// TIA Portal project "bascule_de_controle" (V15)

(* hardware
DEVICE "Station S7-1200_1"  S7-1200 Station
   slot 0: "Châssis_0"  S7-1200 Rack  Rack  V1.0
   slot 1: "PLC_1"  CPU 1215C AC/DC/Rly  6ES7 215-1BG40-0XB0  V4.2
DEVICE "HMI_1"  KTP700 Basic PN
   slot 0: "HMI_1"  KTP700 Basic PN  6AV2 123-2GB03-0AX0  15.0.0.0
   slot 1: "HMI_RT_1"  KTP700 Basic PN  6AV2 123-2GB03-0AX0  15.0.0.0
   slot 5: "HMI_1.IE_CP_1"  PROFINET Interface  15.0.0.0
      slot 1: "Interface PROFINET_1"  PROFINET Interface
         slot 1: "Port_1"  Port
*)

// ===== PLC "PLC_1"  CPU 1215C AC/DC/Rly =====

VAR_GLOBAL   // PLC tag table "Table de variables standard"
   "System_Byte" AT %MB1 : Byte;
   "FirstScan" AT %M1.0 : Bool;
   "DiagStatusUpdate" AT %M1.1 : Bool;
   "AlwaysTRUE" AT %M1.2 : Bool;
   "AlwaysFALSE" AT %M1.3 : Bool;
   "Clock_Byte" AT %MB0 : Byte;
   "Clock_10Hz" AT %M0.0 : Bool;
   "Clock_5Hz" AT %M0.1 : Bool;
   "Clock_2.5Hz" AT %M0.2 : Bool;
   "Clock_2Hz" AT %M0.3 : Bool;
   "Clock_1.25Hz" AT %M0.4 : Bool;
   "Clock_1Hz" AT %M0.5 : Bool;
   "Clock_0.625Hz" AT %M0.6 : Bool;
   "Clock_0.5Hz" AT %M0.7 : Bool;
   "temps_ecoulées" AT %M5.1 : Bool;
   "compter" AT %MW7 : Int;
   "temps_ecoulés" AT %M5.0 : Bool;
   "pesage" AT %MW3 : Word;
   "nbre_bac" AT %MW10 : Int;
   "C_OK" AT %M9.0 : Bool;
   "ENABLE" AT %M9.1 : Bool;
   "depart" AT %Q0.7 : Bool;
END_VAR

VAR_GLOBAL   // PLC tag table "variables_pfa"
   "dcy" AT %I0.0 : Bool;
   "S0" AT %I0.1 : Bool;
   "S1" AT %I0.2 : Bool;
   "EB" AT %I0.3 : Bool;
   "SB" AT %I0.4 : Bool;
   "Tv" AT %I0.5 : Bool;
   "Tf" AT %I0.6 : Bool;
   "C10" AT %I0.7 : Bool;
   "C11" AT %I1.0 : Bool;
   "C20" AT %I1.1 : Bool;
   "C21" AT %I1.2 : Bool;
   "X0" AT %M2.0 : Bool;
   "X1" AT %M2.1 : Bool;
   "X2" AT %M2.2 : Bool;
   "X3" AT %M2.3 : Bool;
   "X4" AT %M2.4 : Bool;
   "X5" AT %M2.5 : Bool;
   "X6" AT %M2.6 : Bool;
   "X7" AT %M2.7 : Bool;
   "X8" AT %M3.0 : Bool;
   "X9" AT %M3.1 : Bool;
   "X10" AT %M3.2 : Bool;
   "X11" AT %M3.3 : Bool;
   "KM1" AT %Q0.0 : Bool;
   "H1" AT %Q0.1 : Bool;
   "BP" AT %Q0.2 : Bool;
   "SV1" AT %Q0.3 : Bool;
   "RV1" AT %Q0.4 : Bool;
   "SV2" AT %Q0.5 : Bool;
   "RV2" AT %Q0.6 : Bool;
   "RA" AT %I1.3 : Bool;
   "alarm_succés" AT %M4.0 : Bool;
   "alarm_error" AT %M4.1 : Bool;
   "alarm" AT %MW5 : Int;
END_VAR

// folder: System blocks/Program resources

DATA_BLOCK "IEC_Timer_0_DB"   // DB1
{ S7_Optimized_Access := 'TRUE' }
AUTHOR : Simatic
FAMILY : IEC
NAME : IEC_TMR
VERSION : 1.0
// stored: InstanceOfName IEC_TIMER
"IEC_TIMER"
BEGIN
END_DATA_BLOCK

DATA_BLOCK "compteur1"   // DB2
{ S7_Optimized_Access := 'TRUE' }
AUTHOR : Simatic
FAMILY : IEC
NAME : CNTR
VERSION : 1.0
// stored: InstanceOfName IEC_COUNTER
"IEC_COUNTER"
BEGIN
END_DATA_BLOCK

// folder: (top level)

FUNCTION "equation_etapes" : Void   // FC1, LAD
{ S7_Optimized_Access := 'TRUE' }
VERSION : 0.1
BEGIN

REGION Network 1: Activation X0
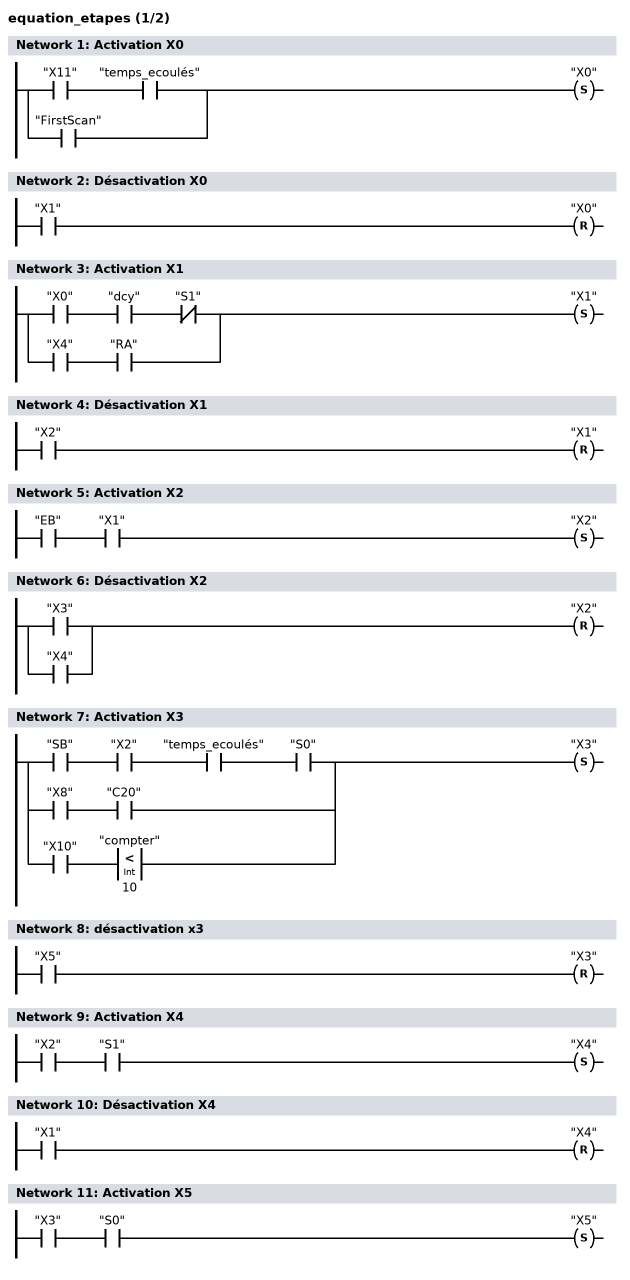
   RUNG wire#powerrail
      Contact( "X11" )
      Contact( "temps_ecoulés" )
      wire#w1
      S_Coil( "X0" )
   END_RUNG
   RUNG wire#powerrail
      Contact( "FirstScan" )
   END_RUNG wire#w1
   // the same network as SCL:
   IF ("X11" AND "temps_ecoulés") OR "FirstScan" THEN "X0" := TRUE; END_IF;
END_REGION

REGION Network 2: Désactivation X0
   RUNG wire#powerrail
      Contact( "X1" )
      R_Coil( "X0" )
   END_RUNG
   // the same network as SCL:
   IF "X1" THEN "X0" := FALSE; END_IF;
END_REGION

REGION Network 3: Activation X1
   RUNG wire#powerrail
      Contact( "X0" )
      Contact( "dcy" )
      I_Contact( "S1" )
      wire#w1
      S_Coil( "X1" )
   END_RUNG
   RUNG wire#powerrail
      Contact( "X4" )
      Contact( "RA" )
   END_RUNG wire#w1
   // the same network as SCL:
   IF ("X0" AND "dcy" AND NOT "S1") OR ("X4" AND "RA") THEN "X1" := TRUE; END_IF;
END_REGION

REGION Network 4: Désactivation X1
   RUNG wire#powerrail
      Contact( "X2" )
      R_Coil( "X1" )
   END_RUNG
   // the same network as SCL:
   IF "X2" THEN "X1" := FALSE; END_IF;
END_REGION

REGION Network 5: Activation X2
   RUNG wire#powerrail
      Contact( "EB" )
      Contact( "X1" )
      S_Coil( "X2" )
   END_RUNG
   // the same network as SCL:
   IF "EB" AND "X1" THEN "X2" := TRUE; END_IF;
END_REGION

REGION Network 6: Désactivation X2
   RUNG wire#powerrail
      Contact( "X3" )
      wire#w1
      R_Coil( "X2" )
   END_RUNG
   RUNG wire#powerrail
      Contact( "X4" )
   END_RUNG wire#w1
   // the same network as SCL:
   IF "X3" OR "X4" THEN "X2" := FALSE; END_IF;
END_REGION

REGION Network 7: Activation X3
   RUNG wire#powerrail
      Contact( "SB" )
      Contact( "X2" )
      Contact( "temps_ecoulés" )
      Contact( "S0" )
      wire#w1
      S_Coil( "X3" )
   END_RUNG
   RUNG wire#powerrail
      Contact( "X8" )
      Contact( "C20" )
   END_RUNG wire#w1
   RUNG wire#powerrail
      Contact( "X10" )
      { S7_Templates := "SrcType := Int" } LT_Contact(in1 := "compter", in2 := 10)
   END_RUNG wire#w1
   // the same network as SCL:
   IF ("SB" AND "X2" AND "temps_ecoulés" AND "S0") OR ("X8" AND "C20") OR ("X10" AND ("compter" < 10)) THEN
       "X3" := TRUE;
   END_IF;
END_REGION

REGION Network 8: désactivation x3
   RUNG wire#powerrail
      Contact( "X5" )
      R_Coil( "X3" )
   END_RUNG
   // the same network as SCL:
   IF "X5" THEN "X3" := FALSE; END_IF;
END_REGION

REGION Network 9: Activation X4
   RUNG wire#powerrail
      Contact( "X2" )
      Contact( "S1" )
      S_Coil( "X4" )
   END_RUNG
   // the same network as SCL:
   IF "X2" AND "S1" THEN "X4" := TRUE; END_IF;
END_REGION

REGION Network 10: Désactivation X4
   RUNG wire#powerrail
      Contact( "X1" )
      R_Coil( "X4" )
   END_RUNG
   // the same network as SCL:
   IF "X1" THEN "X4" := FALSE; END_IF;
END_REGION

REGION Network 11: Activation X5
   RUNG wire#powerrail
      Contact( "X3" )
      Contact( "S0" )
      S_Coil( "X5" )
   END_RUNG
   // the same network as SCL:
   IF "X3" AND "S0" THEN "X5" := TRUE; END_IF;
END_REGION

REGION Network 12: Désactivation X5
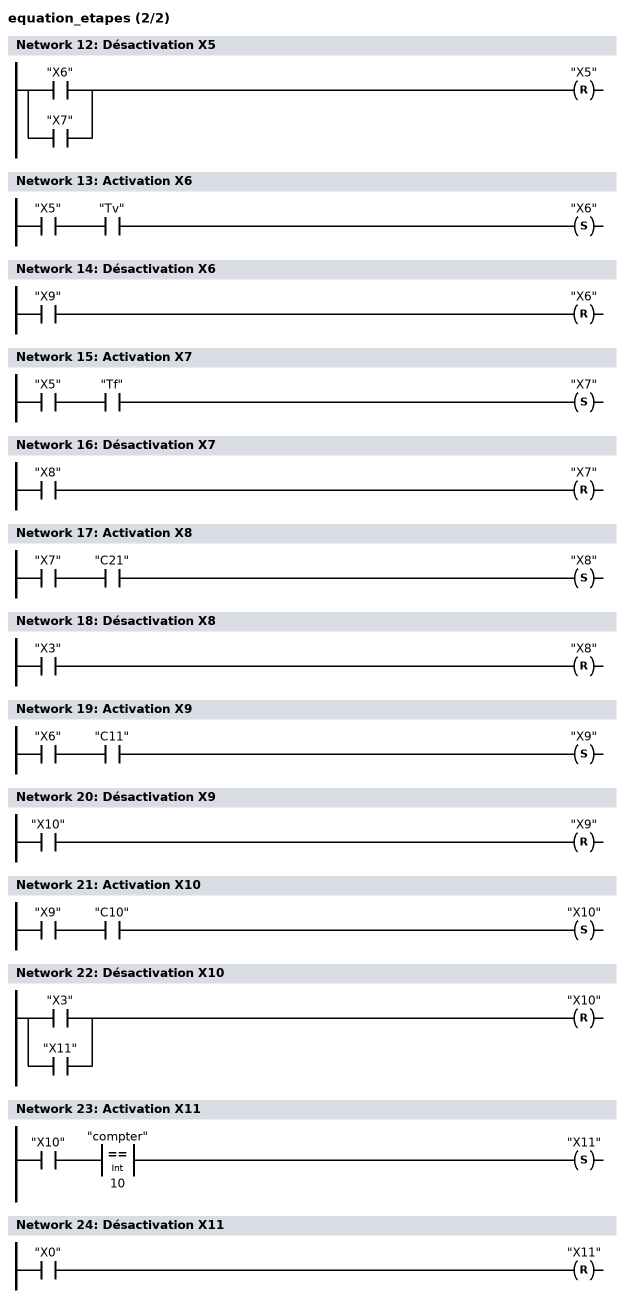
   RUNG wire#powerrail
      Contact( "X6" )
      wire#w1
      R_Coil( "X5" )
   END_RUNG
   RUNG wire#powerrail
      Contact( "X7" )
   END_RUNG wire#w1
   // the same network as SCL:
   IF "X6" OR "X7" THEN "X5" := FALSE; END_IF;
END_REGION

REGION Network 13: Activation X6
   RUNG wire#powerrail
      Contact( "X5" )
      Contact( "Tv" )
      S_Coil( "X6" )
   END_RUNG
   // the same network as SCL:
   IF "X5" AND "Tv" THEN "X6" := TRUE; END_IF;
END_REGION

REGION Network 14: Désactivation X6
   RUNG wire#powerrail
      Contact( "X9" )
      R_Coil( "X6" )
   END_RUNG
   // the same network as SCL:
   IF "X9" THEN "X6" := FALSE; END_IF;
END_REGION

REGION Network 15: Activation X7
   RUNG wire#powerrail
      Contact( "X5" )
      Contact( "Tf" )
      S_Coil( "X7" )
   END_RUNG
   // the same network as SCL:
   IF "X5" AND "Tf" THEN "X7" := TRUE; END_IF;
END_REGION

REGION Network 16: Désactivation X7
   RUNG wire#powerrail
      Contact( "X8" )
      R_Coil( "X7" )
   END_RUNG
   // the same network as SCL:
   IF "X8" THEN "X7" := FALSE; END_IF;
END_REGION

REGION Network 17: Activation X8
   RUNG wire#powerrail
      Contact( "X7" )
      Contact( "C21" )
      S_Coil( "X8" )
   END_RUNG
   // the same network as SCL:
   IF "X7" AND "C21" THEN "X8" := TRUE; END_IF;
END_REGION

REGION Network 18: Désactivation X8
   RUNG wire#powerrail
      Contact( "X3" )
      R_Coil( "X8" )
   END_RUNG
   // the same network as SCL:
   IF "X3" THEN "X8" := FALSE; END_IF;
END_REGION

REGION Network 19: Activation X9
   RUNG wire#powerrail
      Contact( "X6" )
      Contact( "C11" )
      S_Coil( "X9" )
   END_RUNG
   // the same network as SCL:
   IF "X6" AND "C11" THEN "X9" := TRUE; END_IF;
END_REGION

REGION Network 20: Désactivation X9
   RUNG wire#powerrail
      Contact( "X10" )
      R_Coil( "X9" )
   END_RUNG
   // the same network as SCL:
   IF "X10" THEN "X9" := FALSE; END_IF;
END_REGION

REGION Network 21: Activation X10
   RUNG wire#powerrail
      Contact( "X9" )
      Contact( "C10" )
      S_Coil( "X10" )
   END_RUNG
   // the same network as SCL:
   IF "X9" AND "C10" THEN "X10" := TRUE; END_IF;
END_REGION

REGION Network 22: Désactivation X10
   RUNG wire#powerrail
      Contact( "X3" )
      wire#w1
      R_Coil( "X10" )
   END_RUNG
   RUNG wire#powerrail
      Contact( "X11" )
   END_RUNG wire#w1
   // the same network as SCL:
   IF "X3" OR "X11" THEN "X10" := FALSE; END_IF;
END_REGION

REGION Network 23: Activation X11
   RUNG wire#powerrail
      Contact( "X10" )
      { S7_Templates := "SrcType := Int" } EQ_Contact(in1 := "compter", in2 := 10)
      S_Coil( "X11" )
   END_RUNG
   // the same network as SCL:
   IF "X10" AND ("compter" = 10) THEN "X11" := TRUE; END_IF;
END_REGION

REGION Network 24: Désactivation X11
   RUNG wire#powerrail
      Contact( "X0" )
      R_Coil( "X11" )
   END_RUNG
   // the same network as SCL:
   IF "X0" THEN "X11" := FALSE; END_IF;
END_REGION
END_FUNCTION

FUNCTION "les actions" : Void   // FC2, LAD
{ S7_Optimized_Access := 'TRUE' }
VERSION : 0.1
   VAR_TEMP   // added for the SCL form of the ladder/FBD networks
      _w1 : Bool;
   END_VAR
BEGIN

REGION Network 1
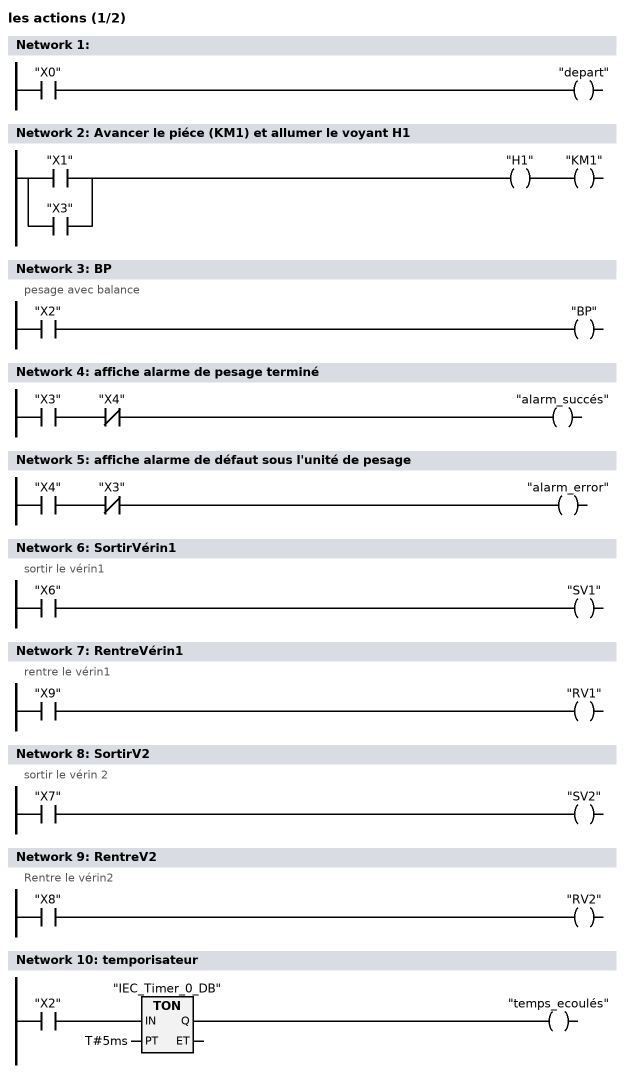
   RUNG wire#powerrail
      Contact( "X0" )
      Coil( "depart" )
   END_RUNG
   // the same network as SCL:
   "depart" := "X0";
END_REGION

REGION Network 2: Avancer le piéce (KM1) et allumer le voyant H1
   RUNG wire#powerrail
      Contact( "X1" )
      wire#w1
      Coil( "H1" )
      Coil( "KM1" )
   END_RUNG
   RUNG wire#powerrail
      Contact( "X3" )
   END_RUNG wire#w1
   // the same network as SCL:
   "H1" := "X1" OR "X3";
   "KM1" := "H1";
END_REGION

REGION Network 3: BP
   // pesage avec balance
   RUNG wire#powerrail
      Contact( "X2" )
      Coil( "BP" )
   END_RUNG
   // the same network as SCL:
   "BP" := "X2";
END_REGION

REGION Network 4: affiche alarme de pesage terminé
   RUNG wire#powerrail
      Contact( "X3" )
      I_Contact( "X4" )
      Coil( "alarm_succés" )
   END_RUNG
   // the same network as SCL:
   "alarm_succés" := "X3" AND NOT "X4";
END_REGION

REGION Network 5: affiche alarme de défaut sous l'unité de pesage
   RUNG wire#powerrail
      Contact( "X4" )
      I_Contact( "X3" )
      Coil( "alarm_error" )
   END_RUNG
   // the same network as SCL:
   "alarm_error" := "X4" AND NOT "X3";
END_REGION

REGION Network 6: SortirVérin1
   // sortir le vérin1
   RUNG wire#powerrail
      Contact( "X6" )
      Coil( "SV1" )
   END_RUNG
   // the same network as SCL:
   "SV1" := "X6";
END_REGION

REGION Network 7: RentreVérin1
   // rentre le vérin1
   RUNG wire#powerrail
      Contact( "X9" )
      Coil( "RV1" )
   END_RUNG
   // the same network as SCL:
   "RV1" := "X9";
END_REGION

REGION Network 8: SortirV2
   // sortir le vérin 2
   RUNG wire#powerrail
      Contact( "X7" )
      Coil( "SV2" )
   END_RUNG
   // the same network as SCL:
   "SV2" := "X7";
END_REGION

REGION Network 9: RentreV2
   // Rentre le vérin2
   RUNG wire#powerrail
      Contact( "X8" )
      Coil( "RV2" )
   END_RUNG
   // the same network as SCL:
   "RV2" := "X8";
END_REGION

REGION Network 10: temporisateur
   "IEC_Timer_0_DB".TON(IN := "X2", PT := T#5ms);
   "temps_ecoulés" := "IEC_Timer_0_DB".Q;
END_REGION

REGION Network 11: compteur des piéces
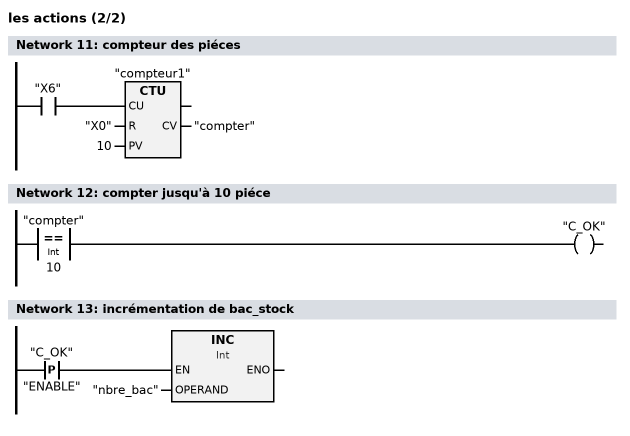
   "compteur1".CTU(CU := "X6", R := "X0", PV := 10, CV => "compter");
END_REGION

REGION Network 12: compter jusqu'à 10 piéce
   RUNG wire#powerrail
      { S7_Templates := "SrcType := Int" } EQ_Contact(in1 := "compter", in2 := 10)
      Coil( "C_OK" )
   END_RUNG
   // the same network as SCL:
   "C_OK" := "compter" = 10;
END_REGION

REGION Network 13: incrémentation de bac_stock
   RUNG wire#powerrail
      P_Contact(operand := "C_OK", bit := "ENABLE")
      { S7_Templates := "DestType := Int" } Inc( "nbre_bac" )
   END_RUNG
   // the same network as SCL:
   #_w1 := "C_OK" AND NOT "ENABLE";   // rising edge of "C_OK"
   "ENABLE" := "C_OK";
   IF #_w1 THEN "nbre_bac" := "nbre_bac" + 1; END_IF;
END_REGION
END_FUNCTION

ORGANIZATION_BLOCK "Main"   // OB1, LAD, ProgramCycle
TITLE = "Main Program Sweep (Cycle)"
{ S7_Optimized_Access := 'TRUE' }
VERSION : 0.1
   VAR_INPUT
      Initial_Call : Bool;   // Initial call of this OB
      Remanence : Bool;   // =True, if remanent data are available
   END_VAR
BEGIN

REGION Network 1
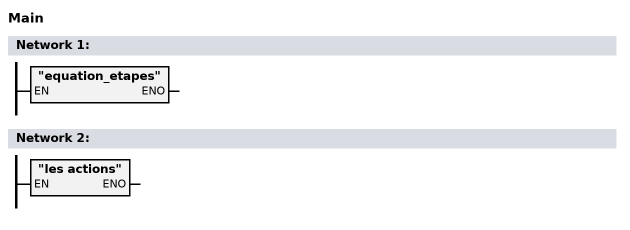
   RUNG wire#powerrail
      "equation_etapes"()
   END_RUNG
   // the same network as SCL:
   "equation_etapes"();
END_REGION

REGION Network 2
   RUNG wire#powerrail
      "les actions"()
   END_RUNG
   // the same network as SCL:
   "les actions"();
END_REGION
END_ORGANIZATION_BLOCK

(* ===== HMI "HMI_RT_1" =====
system functions are stored by id; their names below are inferred from use
connection "HMI_Liaison_1": ETHERNET, SMART_S7_1200_OMS

HMI tags "Table de variables standard"
   "alarm" : Word = PLC pesage AT %MW3, 1 s
   "voyant" : Bool = PLC H1 AT %Q0.1, 1 s
   "Variable_IHM_1" : Int = PLC compter AT %MW7, 1 s
   "Variable_IHM_1(1)" : Int = PLC nbre_bac AT %MW10, 1 s
   "Variable_IHM_1(2)" : Bool = PLC dcy AT %I0.0, 1 s
   "depart" : Bool = PLC FirstScan AT %M1.0, 1 s
   "Variable_IHM_1(3)" : Bool = PLC FirstScan AT %M1.0, 1 s
   "Variable_IHM_1(4)" : Bool = PLC depart AT %Q0.7, 1 s
   "X0" : Bool = PLC X0 AT %M2.0, 1 s

discrete alarms
   1: 'pesage terminé avec succés', class alarm_pesage, trigger "alarm" bit 0
   2: 'pesage echoué', class alarm_pesage, trigger "alarm" bit 1

text list "Nom_vue_liste_textes": 1 'Vue racine'

Template "Modèle_1" 800x480
   Button "Template_Button" at 375,727 size 50x71; TextOff 'Text'
   Button "Template_Button_1" at 321,727 size 50x71; TextOff 'Text'
   Button "Template_Button_2" at 268,727 size 50x71; TextOff 'Text'
   Button "Template_Button_3" at 214,727 size 50x71; TextOff 'Text'
   Button "Template_Button_4" at 161,727 size 50x71; TextOff 'Text'
   Button "Template_Button_5" at 108,727 size 50x71; TextOff 'Text'
   Button "Template_Button_6" at 54,727 size 50x71; TextOff 'Text'
   Button "Vue initiale" at 1,727 size 50x71; TextOff 'Vue initiale'; PictureOff "NavigateHome_KTP700_Basic_PN_Portrait_TR"; PictureOn "NavigateHome_KTP700_Basic_PN_Portrait_TR"
      on Release: ActivateScreen("principale", 0)
   Button "Quitter" at 428,727 size 50x71; TextOff 'Quitter'; PictureOff "ExitRuntime_KTP700_Basic_PN_Portrait_TR"; PictureOn "ExitRuntime_KTP700_Basic_PN_Portrait_TR"
      on Release: StopRuntime(0)
   SymbolicIOField "Vue_champ_ES_symbolique" at 109,11 size 264x38; TextOff '0'; TextOn '1'; TextList "Nom_vue_liste_textes"
      ProcessValue <- "alarm"
      on Change: ActivateScreenByNumber("alarm", 0)
   DateTimeField "HmiScreenItemData" at 375,30 size 105x30
   DateTimeField "HmiScreenItemData_1" at 375,0 size 105x30
   GraphicView "Logo" at 0,0 size 107x60; Picture "Logo de HMI_1"

screen "principale" 800x480, template "Modèle_1"
   on GenerateScreen: SetTag("alarm", 1)
   Circle "Cercle_1" at 175,152 size 80x80
      Appearance <- "Variable_IHM_1(4)"
   TextField "Champ de texte_1" at 628,0 size 160x34; Text 'May Nesrine'
   Button "Bouton_1" at 344,120 size 291x67; TextOff 'Alarme'
      on Click: ActivateScreen("Alarme", 0)
   Button "Bouton_2" at 344,241 size 290x61; TextOff 'Supervision'
      on Click: ActivateScreen("Supervision", 0)
   TextField "Champ de texte_2" at 83,110 size 136x23; Text 'départ_systéme'
   TextField "Champ de texte_3" at 119,11 size 248x33; Text 'Bascule de controle'
   Switch "Commutateur_1" at 30,166 size 123x59; CaptionText 'Switch'; TextOff 'OFF'; TextOn 'ON'
      ProcessValue <- "X0"

screen "Alarme" 800x480
   TextField "Champ de texte_1" at 7,9 size 204x29; Text 'Alarme_de_pesage'
   DateTimeField "Champ de date/heure_1" at 491,13 size 188x32
   AlarmView "Vue des alarmes_1" at 11,91 size 718x314
   Button "Bouton_1" at 68,409 size 353x51; TextOff 'Principale'
      on Click: ActivateScreen("principale", 0)

screen "Supervision" 800x480
   TextField "Champ de texte_1" at 39,17 size 232x27; Text 'Supervision du systéme'
   DateTimeField "Champ de date/heure_1" at 528,20 size 188x32
   TextField "Champ de texte_2" at 454,278 size 191x37; Text 'bac_de_stock'
   GraphicView "Vue de graphique_1" at 271,231 size 204x133; Picture "Graphique_1"
   IOField "Champ d'E/S_1" at 196,292 size 101x34; FormatPattern s99999
      ProcessValue <- "Variable_IHM_1(1)"
   IOField "Champ d'E/S_2" at 251,145 size 99x34; FormatPattern s99
      ProcessValue <- "Variable_IHM_1"
   TextField "Champ de texte_3" at 12,142 size 229x35; Text 'nbre_des_piéces'
   Button "Bouton_1" at 49,380 size 192x32; TextOff 'principale'
      on Click: ActivateScreen("principale", 0)
   TextField "Champ de texte_4" at 318,292 size 81x23; Text '10 piéces'
   Circle "Cercle_1" at 633,68 size 57x57
      Appearance <- "voyant"
   TextField "Champ de texte_5" at 475,80 size 158x25; Text 'Tapis_en_avance'
*)